FUNCTION_BLOCK FB_MachineControl
VAR_INPUT
END_VAR
VAR_OUTPUT
END_VAR
VAR
END_VAR

END_FUNCTION_BLOCK

(* stored: Version 1.1.0.1
   POU FB_MachineControl: Id {67dc6557-4e18-4480-9e46-d86d55fce5be}, SpecialFunc None *)
